TYPE ItemState :
STRUCT
	InProcess	:	BOOL;			// item picked-up by robot & processing by workcenter 
	Done		:	BOOL;			// item processing completed
END_STRUCT
END_TYPE

(* stored: Version 1.1.0.1, ProductVersion 3.1.4024.15
   DUT ItemState: Id {e9743a97-0fef-4dd2-b36e-85c1ff9bbcb6} *)
